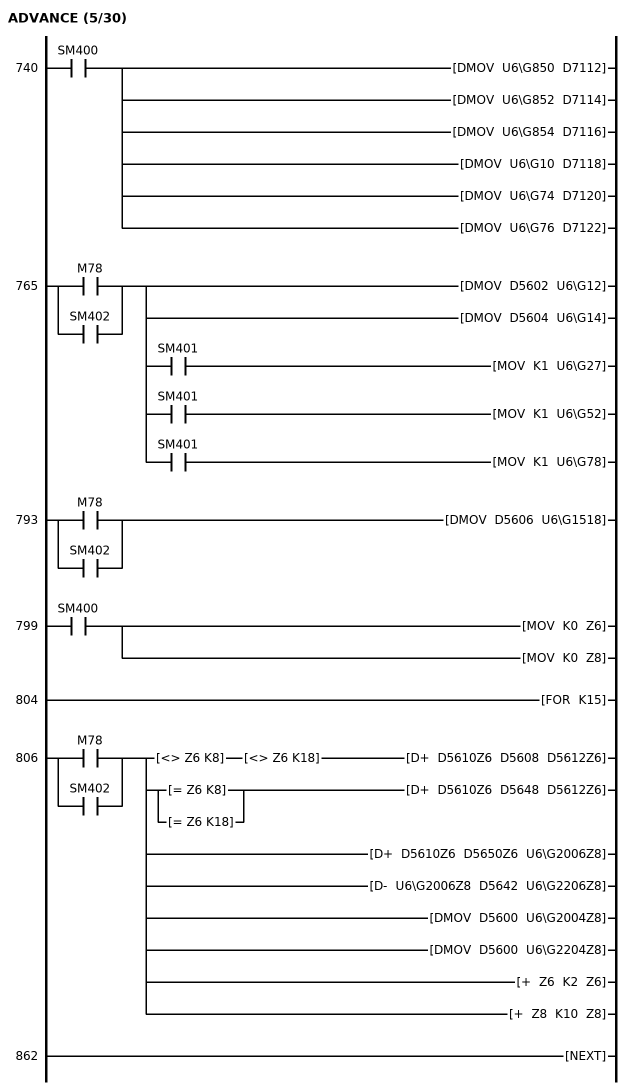
[picture p360: ladder of ADVANCE, rungs at steps 740 to 862]
740   LD      SM400
      DMOV    U6\G850 D7112
      DMOV    U6\G852 D7114
      DMOV    U6\G854 D7116
      DMOV    U6\G10 D7118
      DMOV    U6\G74 D7120
      DMOV    U6\G76 D7122
765   LD      M78
      OR      SM402
      DMOV    D5602 U6\G12
      DMOV    D5604 U6\G14
      MPS
      AND     SM401
      MOV     K1 U6\G27
      MRD
      AND     SM401
      MOV     K1 U6\G52
      MPP
      AND     SM401
      MOV     K1 U6\G78
793   LD      M78
      OR      SM402
      DMOV    D5606 U6\G1518
799   LD      SM400
      MOV     K0 Z6
      MOV     K0 Z8
804   FOR     K15
806   LD      M78
      OR      SM402
      MPS
      AND<>   Z6 K8
      AND<>   Z6 K18
      D+      D5610Z6 D5608 D5612Z6
      MRD
      LD=     Z6 K8
      OR=     Z6 K18
      ANB
      D+      D5610Z6 D5648 D5612Z6
      MPP
      D+      D5610Z6 D5650Z6 U6\G2006Z8
      D-      U6\G2006Z8 D5642 U6\G2206Z8
      DMOV    D5600 U6\G2004Z8
      DMOV    D5600 U6\G2204Z8
      +       Z6 K2 Z6
      +       Z8 K10 Z8
862   NEXT
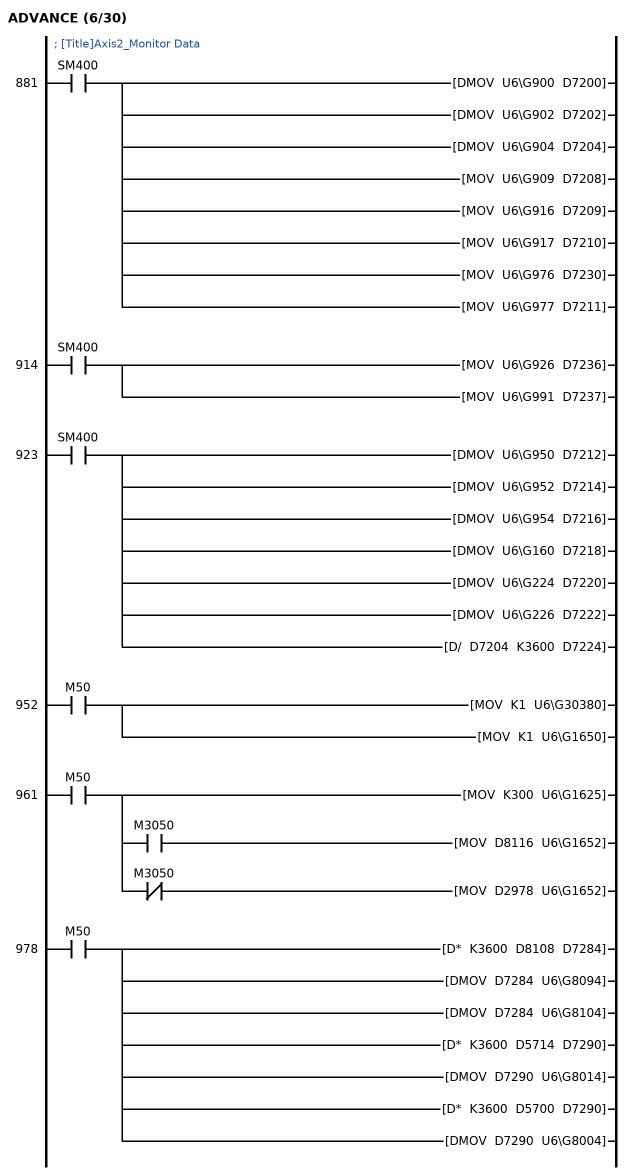
; 
; [Title]Axis2_Monitor Data
; 
; 
881   LD      SM400
      DMOV    U6\G900 D7200
      DMOV    U6\G902 D7202
      DMOV    U6\G904 D7204
      MOV     U6\G909 D7208
      MOV     U6\G916 D7209
      MOV     U6\G917 D7210
      MOV     U6\G976 D7230
      MOV     U6\G977 D7211
914   LD      SM400
      MOV     U6\G926 D7236
      MOV     U6\G991 D7237
923   LD      SM400
      DMOV    U6\G950 D7212
      DMOV    U6\G952 D7214
      DMOV    U6\G954 D7216
      DMOV    U6\G160 D7218
      DMOV    U6\G224 D7220
      DMOV    U6\G226 D7222
      D/      D7204 K3600 D7224
952   LD      M50
      MOV     K1 U6\G30380
      MOV     K1 U6\G1650
961   LD      M50
      MOV     K300 U6\G1625
      MPS
      AND     M3050
      MOV     D8116 U6\G1652
      MPP
      ANI     M3050
      MOV     D2978 U6\G1652
978   LD      M50
      D*      K3600 D8108 D7284
      DMOV    D7284 U6\G8094
      DMOV    D7284 U6\G8104
      D*      K3600 D5714 D7290
      DMOV    D7290 U6\G8014
      D*      K3600 D5700 D7290
      DMOV    D7290 U6\G8004
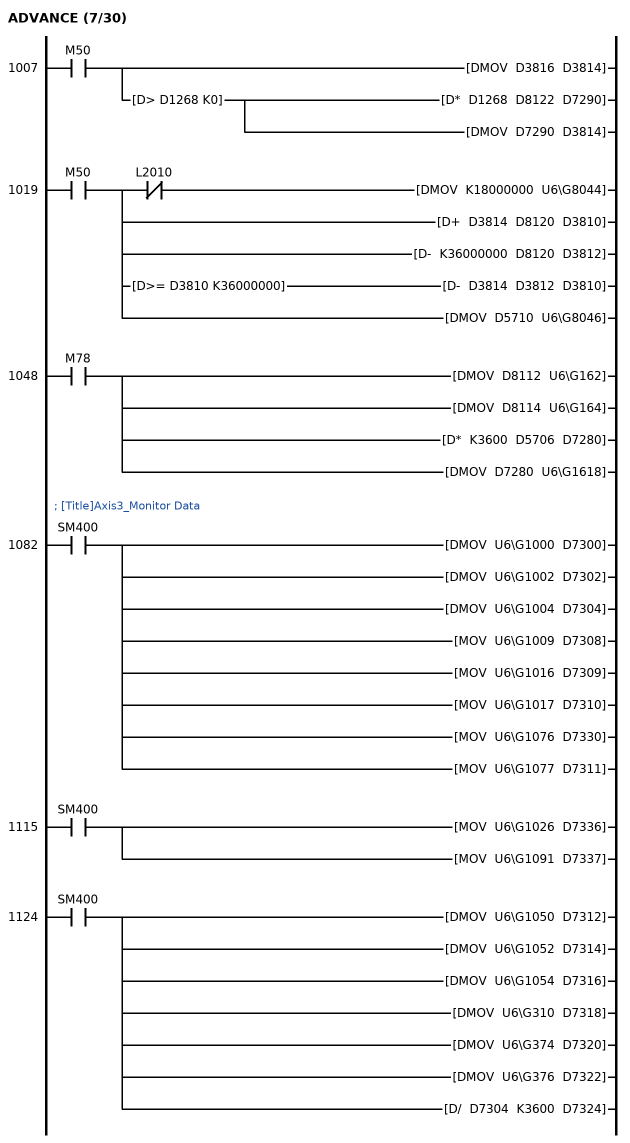
1007  LD      M50
      DMOV    D3816 D3814
      ANDD>   D1268 K0
      D*      D1268 D8122 D7290
      DMOV    D7290 D3814
1019  LD      M50
      MPS
      ANI     L2010
      DMOV    K18000000 U6\G8044
      MPP
      D+      D3814 D8120 D3810
      D-      K36000000 D8120 D3812
      MPS
      ANDD>=  D3810 K36000000
      D-      D3814 D3812 D3810
      MPP
      DMOV    D5710 U6\G8046
1048  LD      M78
      DMOV    D8112 U6\G162
      DMOV    D8114 U6\G164
      D*      K3600 D5706 D7280
      DMOV    D7280 U6\G1618
; 
; [Title]Axis3_Monitor Data
; 
1082  LD      SM400
      DMOV    U6\G1000 D7300
      DMOV    U6\G1002 D7302
      DMOV    U6\G1004 D7304
      MOV     U6\G1009 D7308
      MOV     U6\G1016 D7309
      MOV     U6\G1017 D7310
      MOV     U6\G1076 D7330
      MOV     U6\G1077 D7311
1115  LD      SM400
      MOV     U6\G1026 D7336
      MOV     U6\G1091 D7337
1124  LD      SM400
      DMOV    U6\G1050 D7312
      DMOV    U6\G1052 D7314
      DMOV    U6\G1054 D7316
      DMOV    U6\G310 D7318
      DMOV    U6\G374 D7320
      DMOV    U6\G376 D7322
      D/      D7304 K3600 D7324
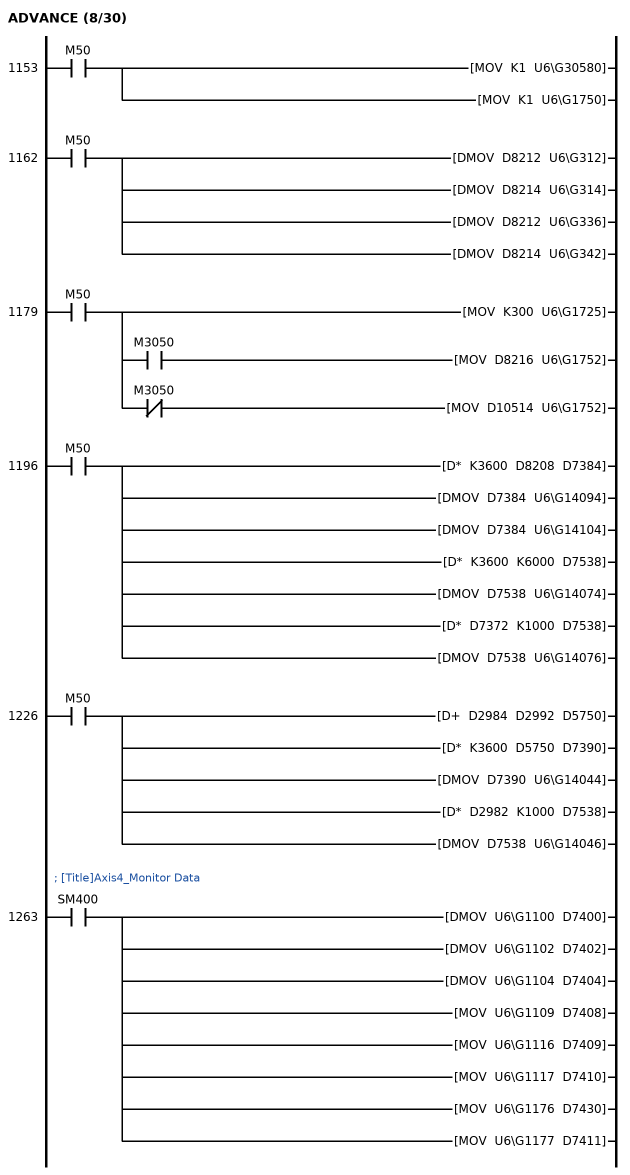
1153  LD      M50
      MOV     K1 U6\G30580
      MOV     K1 U6\G1750
1162  LD      M50
      DMOV    D8212 U6\G312
      DMOV    D8214 U6\G314
      DMOV    D8212 U6\G336
      DMOV    D8214 U6\G342
1179  LD      M50
      MOV     K300 U6\G1725
      MPS
      AND     M3050
      MOV     D8216 U6\G1752
      MPP
      ANI     M3050
      MOV     D10514 U6\G1752
1196  LD      M50
      D*      K3600 D8208 D7384
      DMOV    D7384 U6\G14094
      DMOV    D7384 U6\G14104
      D*      K3600 K6000 D7538
      DMOV    D7538 U6\G14074
      D*      D7372 K1000 D7538
      DMOV    D7538 U6\G14076
1226  LD      M50
      D+      D2984 D2992 D5750
      D*      K3600 D5750 D7390
      DMOV    D7390 U6\G14044
      D*      D2982 K1000 D7538
      DMOV    D7538 U6\G14046
; [Title]Axis4_Monitor Data
; 
; 
1263  LD      SM400
      DMOV    U6\G1100 D7400
      DMOV    U6\G1102 D7402
      DMOV    U6\G1104 D7404
      MOV     U6\G1109 D7408
      MOV     U6\G1116 D7409
      MOV     U6\G1117 D7410
      MOV     U6\G1176 D7430
      MOV     U6\G1177 D7411
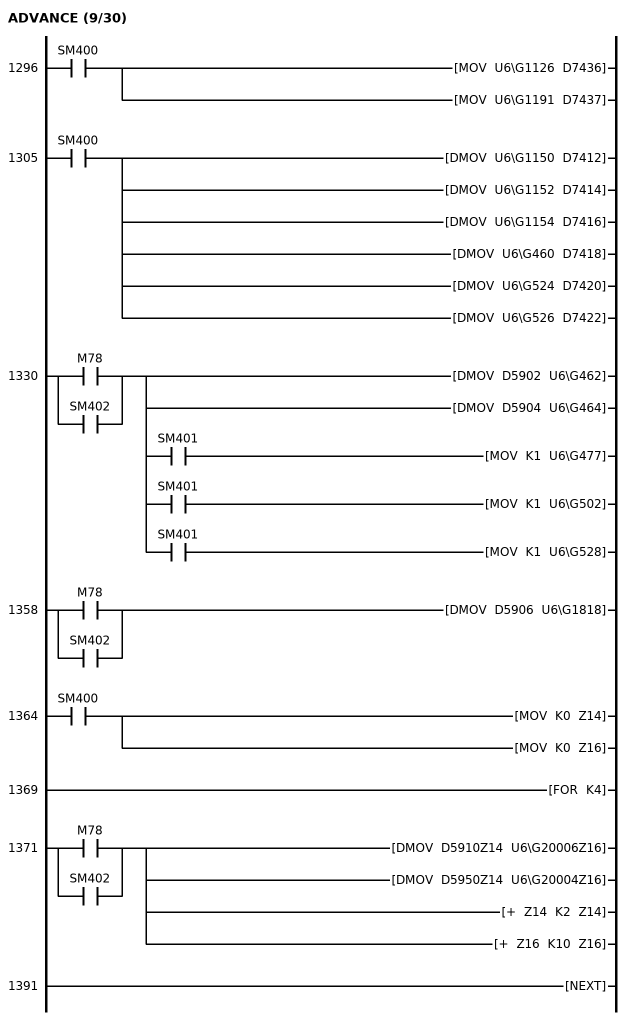
1296  LD      SM400
      MOV     U6\G1126 D7436
      MOV     U6\G1191 D7437
1305  LD      SM400
      DMOV    U6\G1150 D7412
      DMOV    U6\G1152 D7414
      DMOV    U6\G1154 D7416
      DMOV    U6\G460 D7418
      DMOV    U6\G524 D7420
      DMOV    U6\G526 D7422
1330  LD      M78
      OR      SM402
      DMOV    D5902 U6\G462
      DMOV    D5904 U6\G464
      MPS
      AND     SM401
      MOV     K1 U6\G477
      MRD
      AND     SM401
      MOV     K1 U6\G502
      MPP
      AND     SM401
      MOV     K1 U6\G528
1358  LD      M78
      OR      SM402
      DMOV    D5906 U6\G1818
1364  LD      SM400
      MOV     K0 Z14
      MOV     K0 Z16
1369  FOR     K4
1371  LD      M78
      OR      SM402
      DMOV    D5910Z14 U6\G20006Z16
      DMOV    D5950Z14 U6\G20004Z16
      +       Z14 K2 Z14
      +       Z16 K10 Z16
1391  NEXT
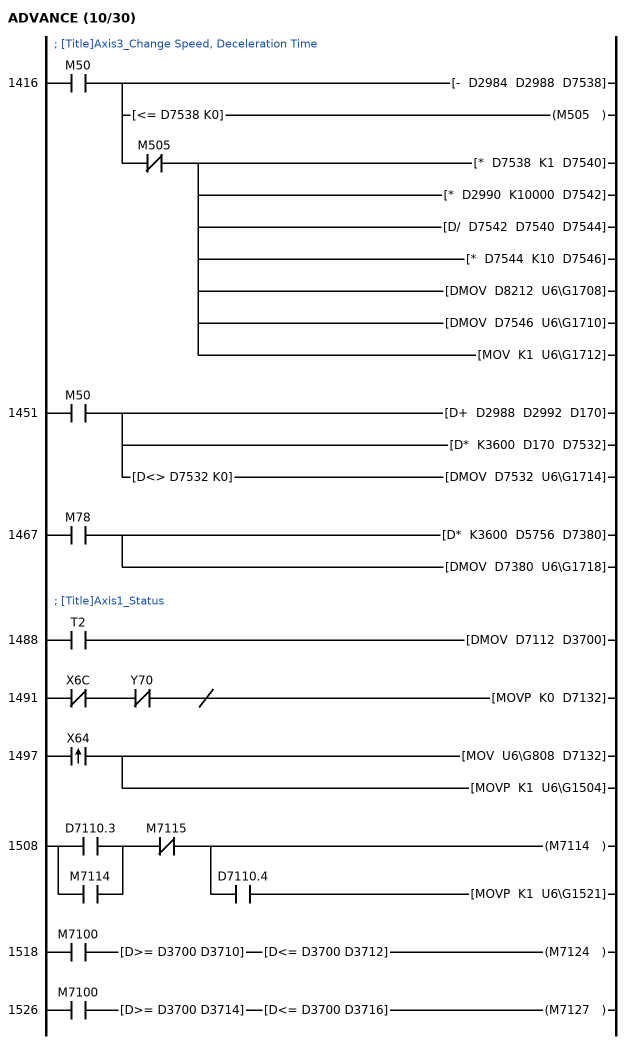
; [Title]Axis3_Change Speed, Deceleration Time
1416  LD      M50
      -       D2984 D2988 D7538
      MPS
      AND<=   D7538 K0
      OUT     M505
      MPP
      ANI     M505
      *       D7538 K1 D7540
      *       D2990 K10000 D7542
      D/      D7542 D7540 D7544
      *       D7544 K10 D7546
      DMOV    D8212 U6\G1708
      DMOV    D7546 U6\G1710
      MOV     K1 U6\G1712
1451  LD      M50
      D+      D2988 D2992 D170
      D*      K3600 D170 D7532
      ANDD<>  D7532 K0
      DMOV    D7532 U6\G1714
1467  LD      M78
      D*      K3600 D5756 D7380
      DMOV    D7380 U6\G1718
; [Title]Axis1_Status
1488  LD      T2
      DMOV    D7112 D3700
1491  LDI     X6C
      ANI     Y70
      INV
      MOVP    K0 D7132
1497  LDP     X64
      MOV     U6\G808 D7132
      MOVP    K1 U6\G1504
1508  LD      D7110.3
      OR      M7114
      ANI     M7115
      OUT     M7114
      AND     D7110.4
      MOVP    K1 U6\G1521
1518  LD      M7100
      ANDD>=  D3700 D3710
      ANDD<=  D3700 D3712
      OUT     M7124
1526  LD      M7100
      ANDD>=  D3700 D3714
      ANDD<=  D3700 D3716
      OUT     M7127
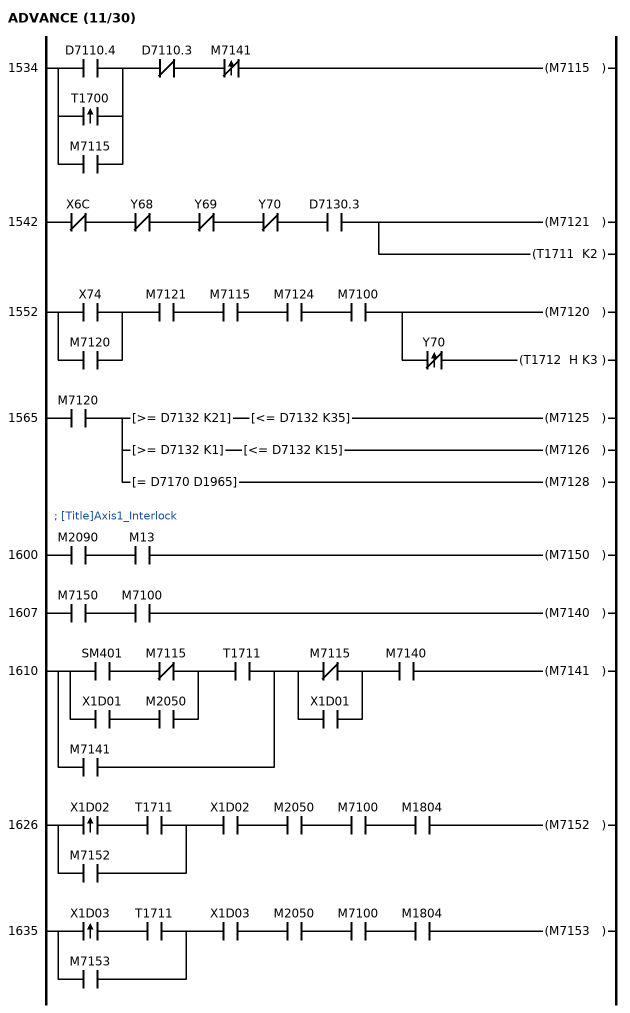
1534  LD      D7110.4
      ORP     T1700
      OR      M7115
      ANI     D7110.3
      ANDPI   M7141
      OUT     M7115
1542  LDI     X6C
      ANI     Y68
      ANI     Y69
      ANI     Y70
      AND     D7130.3
      OUT     M7121
      OUT     T1711 K2
1552  LD      X74
      OR      M7120
      AND     M7121
      AND     M7115
      AND     M7124
      AND     M7100
      OUT     M7120
      ANDPI   Y70
      OUTH    T1712 K3
1565  LD      M7120
      MPS
      AND>=   D7132 K21
      AND<=   D7132 K35
      OUT     M7125
      MRD
      AND>=   D7132 K1
      AND<=   D7132 K15
      OUT     M7126
      MPP
      AND=    D7170 D1965
      OUT     M7128
; [Title]Axis1_Interlock
1600  LD      M2090
      AND     M13
      OUT     M7150
; 
; 
; 
; 
1607  LD      M7150
      AND     M7100
      OUT     M7140
1610  LD      SM401
      ANI     M7115
      LD      X1D01
      AND     M2050
      ORB
      AND     T1711
      OR      M7141
      LDI     M7115
      OR      X1D01
      ANB
      AND     M7140
      OUT     M7141
; 
; 
; 
; 
1626  LDP     X1D02
      AND     T1711
      OR      M7152
      AND     X1D02
      AND     M2050
      AND     M7100
      AND     M1804
      OUT     M7152
1635  LDP     X1D03
      AND     T1711
      OR      M7153
      AND     X1D03
      AND     M2050
      AND     M7100
      AND     M1804
      OUT     M7153
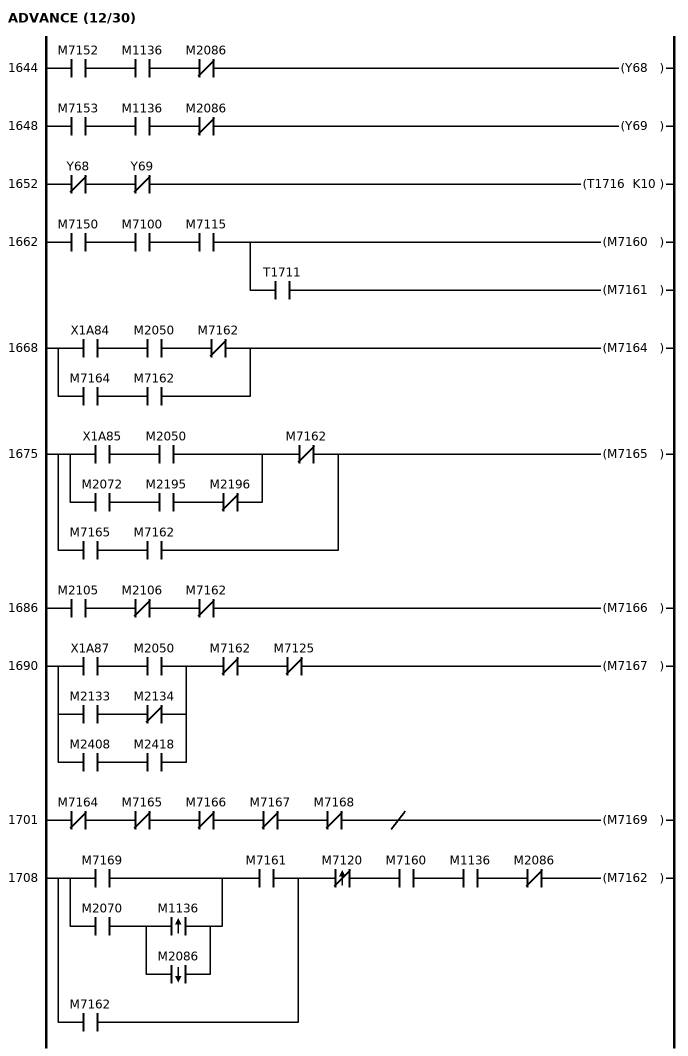
1644  LD      M7152
      AND     M1136
      ANI     M2086
      OUT     Y68
1648  LD      M7153
      AND     M1136
      ANI     M2086
      OUT     Y69
1652  LDI     Y68
      ANI     Y69
      OUT     T1716 K10
; 
; 
; 
; 
1662  LD      M7150
      AND     M7100
      AND     M7115
      OUT     M7160
      AND     T1711
      OUT     M7161
1668  LD      X1A84
      AND     M2050
      ANI     M7162
      LD      M7164
      AND     M7162
      ORB
      OUT     M7164
1675  LD      X1A85
      AND     M2050
      LD      M2072
      AND     M2195
      ANI     M2196
      ORB
      ANI     M7162
      LD      M7165
      AND     M7162
      ORB
      OUT     M7165
1686  LD      M2105
      ANI     M2106
      ANI     M7162
      OUT     M7166
1690  LD      X1A87
      AND     M2050
      LD      M2133
      ANI     M2134
      ORB
      LD      M2408
      AND     M2418
      ORB
      ANI     M7162
      ANI     M7125
      OUT     M7167
1701  LDI     M7164
      ANI     M7165
      ANI     M7166
      ANI     M7167
      ANI     M7168
      INV
      OUT     M7169
1708  LD      M7169
      LD      M2070
      LDP     M1136
      ORF     M2086
      ANB
      ORB
      AND     M7161
      OR      M7162
      ANDPI   M7120
      AND     M7160
      AND     M1136
      ANI     M2086
      OUT     M7162
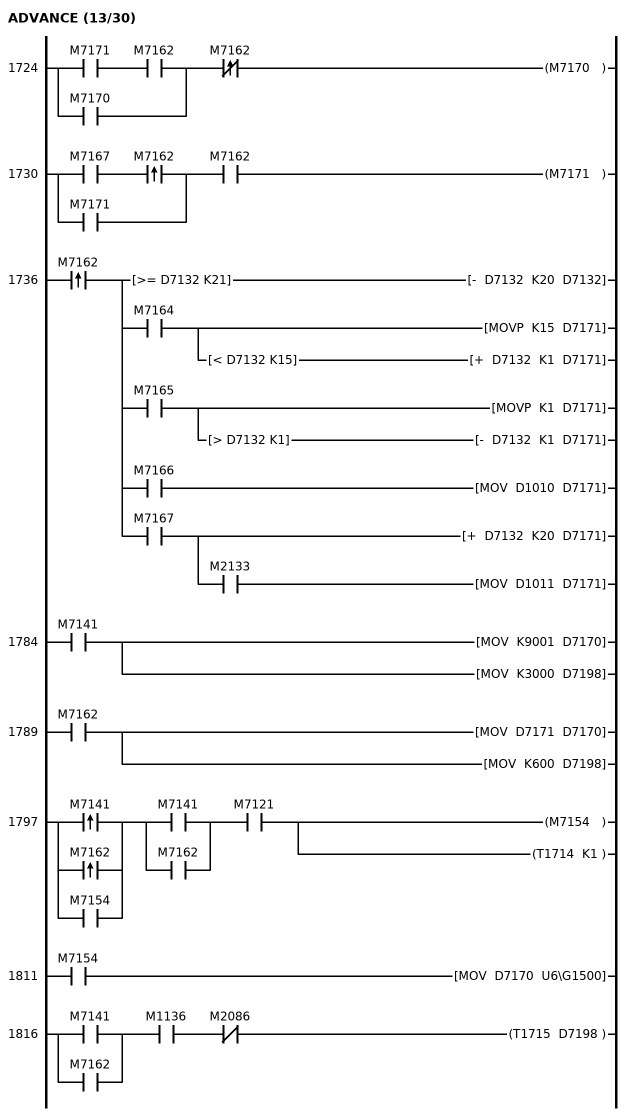
1724  LD      M7171
      AND     M7162
      OR      M7170
      ANDPI   M7162
      OUT     M7170
1730  LD      M7167
      ANDP    M7162
      OR      M7171
      AND     M7162
      OUT     M7171
1736  LDP     M7162
      MPS
      AND>=   D7132 K21
      -       D7132 K20 D7132
      MRD
      AND     M7164
      MOVP    K15 D7171
      AND<    D7132 K15
      +       D7132 K1 D7171
      MRD
      AND     M7165
      MOVP    K1 D7171
      AND>    D7132 K1
      -       D7132 K1 D7171
      MRD
      AND     M7166
      MOV     D1010 D7171
      MPP
      AND     M7167
      +       D7132 K20 D7171
      AND     M2133
      MOV     D1011 D7171
; 
; 
; 
; 
1784  LD      M7141
      MOV     K9001 D7170
      MOV     K3000 D7198
1789  LD      M7162
      MOV     D7171 D7170
      MOV     K600 D7198
; 
; 
; 
1797  LDP     M7141
      ORP     M7162
      OR      M7154
      LD      M7141
      OR      M7162
      ANB
      AND     M7121
      OUT     M7154
      OUT     T1714 K1
1811  LD      M7154
      MOV     D7170 U6\G1500
1816  LD      M7141
      OR      M7162
      AND     M1136
      ANI     M2086
      OUT     T1715 D7198
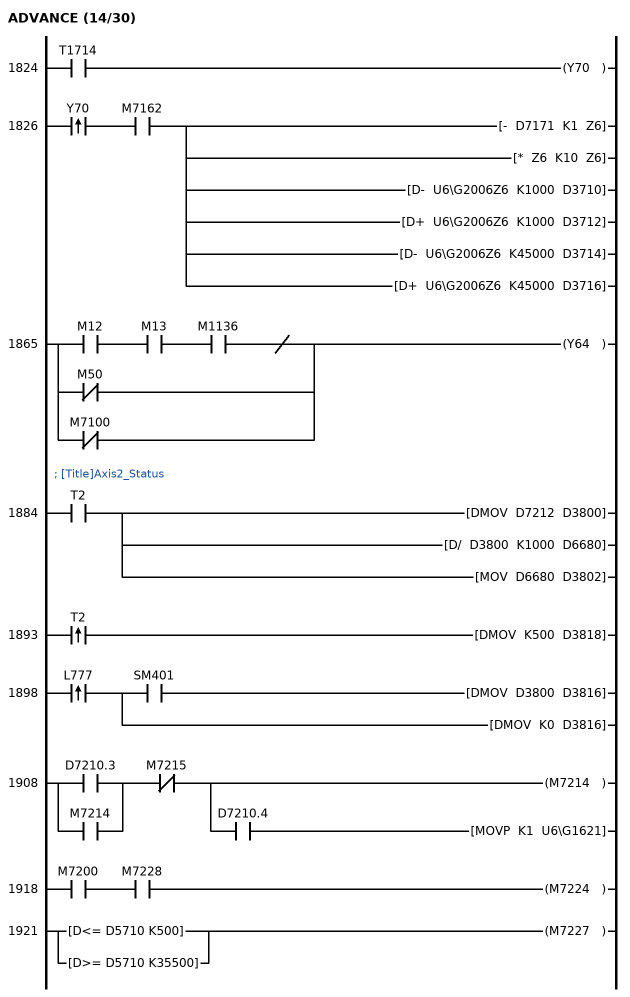
1824  LD      T1714
      OUT     Y70
1826  LDP     Y70
      AND     M7162
      -       D7171 K1 Z6
      *       Z6 K10 Z6
      D-      U6\G2006Z6 K1000 D3710
      D+      U6\G2006Z6 K1000 D3712
      D-      U6\G2006Z6 K45000 D3714
      D+      U6\G2006Z6 K45000 D3716
; 
; 
; 
1865  LD      M12
      AND     M13
      AND     M1136
      INV
      ORI     M50
      ORI     M7100
      OUT     Y64
; [Title]Axis2_Status
1884  LD      T2
      DMOV    D7212 D3800
      D/      D3800 K1000 D6680
      MOV     D6680 D3802
1893  LDP     T2
      DMOV    K500 D3818
1898  LDP     L777
      MPS
      AND     SM401
      DMOV    D3800 D3816
      MPP
      DMOV    K0 D3816
1908  LD      D7210.3
      OR      M7214
      ANI     M7215
      OUT     M7214
      AND     D7210.4
      MOVP    K1 U6\G1621
1918  LD      M7200
      AND     M7228
      OUT     M7224
1921  LDD<=   D5710 K500
      ORD>=   D5710 K35500
      OUT     M7227
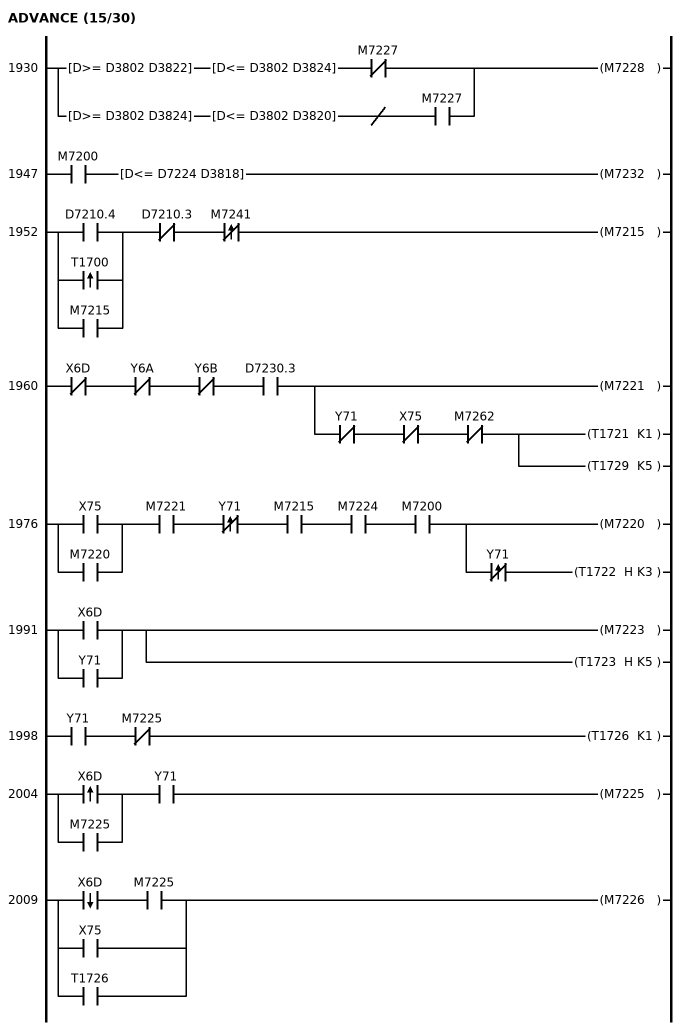
1930  LDD>=   D3802 D3822
      ANDD<=  D3802 D3824
      ANI     M7227
      LDD>=   D3802 D3824
      ANDD<=  D3802 D3820
      INV
      AND     M7227
      ORB
      OUT     M7228
1947  LD      M7200
      ANDD<=  D7224 D3818
      OUT     M7232
1952  LD      D7210.4
      ORP     T1700
      OR      M7215
      ANI     D7210.3
      ANDPI   M7241
      OUT     M7215
1960  LDI     X6D
      ANI     Y6A
      ANI     Y6B
      AND     D7230.3
      OUT     M7221
      ANI     Y71
      ANI     X75
      ANI     M7262
      OUT     T1721 K1
      OUT     T1729 K5
1976  LD      X75
      OR      M7220
      AND     M7221
      ANDPI   Y71
      AND     M7215
      AND     M7224
      AND     M7200
      OUT     M7220
      ANDPI   Y71
      OUTH    T1722 K3
1991  LD      X6D
      OR      Y71
      OUT     M7223
      OUTH    T1723 K5
1998  LD      Y71
      ANI     M7225
      OUT     T1726 K1
2004  LDP     X6D
      OR      M7225
      AND     Y71
      OUT     M7225
2009  LDF     X6D
      AND     M7225
      OR      X75
      OR      T1726
      OUT     M7226
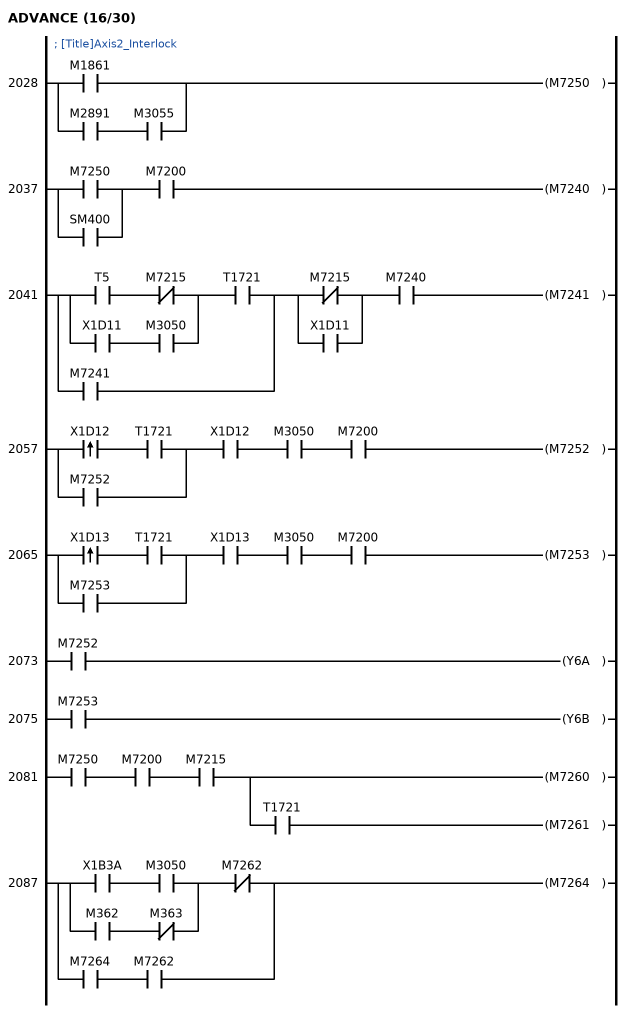
; [Title]Axis2_Interlock
2028  LD      M1861
      LD      M2891
      AND     M3055
      ORB
      OUT     M7250
; 
; 
; 
; 
2037  LD      M7250
      OR      SM400
      AND     M7200
      OUT     M7240
2041  LD      T5
      ANI     M7215
      LD      X1D11
      AND     M3050
      ORB
      AND     T1721
      OR      M7241
      LDI     M7215
      OR      X1D11
      ANB
      AND     M7240
      OUT     M7241
; 
; 
; 
; 
2057  LDP     X1D12
      AND     T1721
      OR      M7252
      AND     X1D12
      AND     M3050
      AND     M7200
      OUT     M7252
2065  LDP     X1D13
      AND     T1721
      OR      M7253
      AND     X1D13
      AND     M3050
      AND     M7200
      OUT     M7253
2073  LD      M7252
      OUT     Y6A
2075  LD      M7253
      OUT     Y6B
; 
; 
; 
; 
2081  LD      M7250
      AND     M7200
      AND     M7215
      OUT     M7260
      AND     T1721
      OUT     M7261
2087  LD      X1B3A
      AND     M3050
      LD      M362
      ANI     M363
      ORB
      ANI     M7262
      LD      M7264
      AND     M7262
      ORB
      OUT     M7264
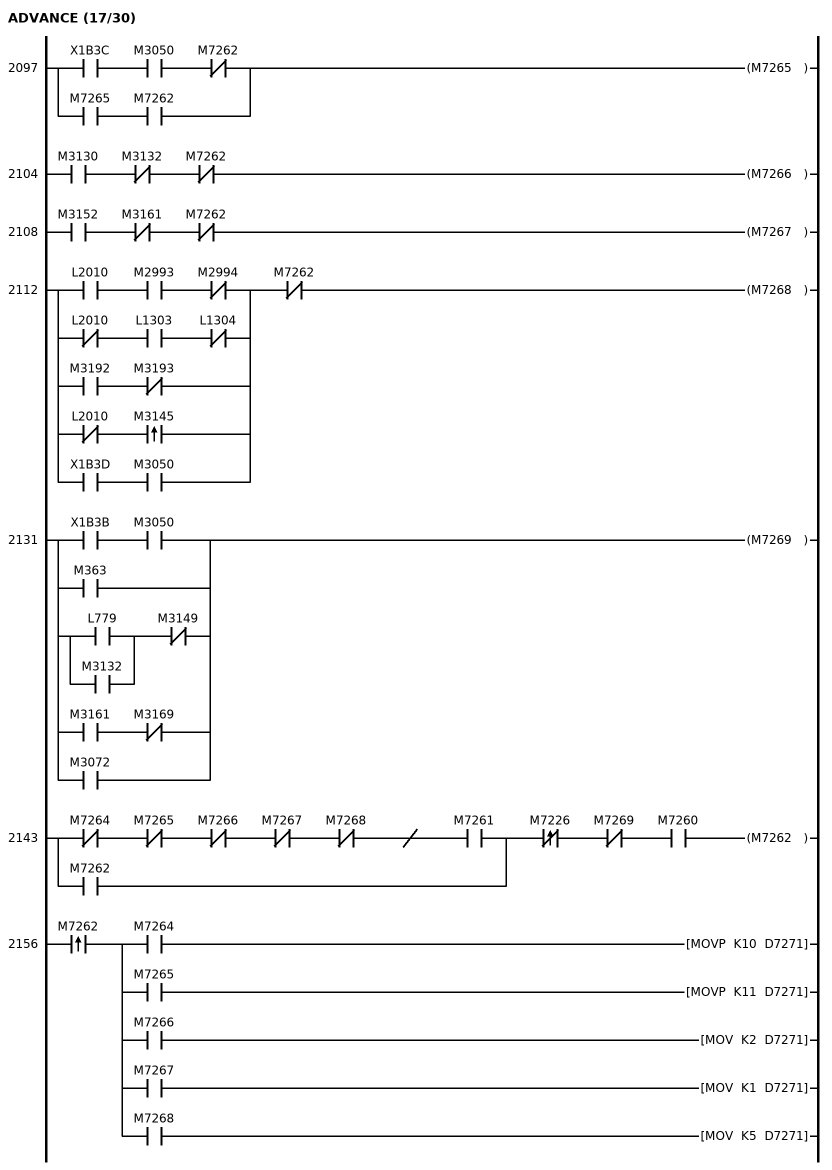
2097  LD      X1B3C
      AND     M3050
      ANI     M7262
      LD      M7265
      AND     M7262
      ORB
      OUT     M7265
2104  LD      M3130
      ANI     M3132
      ANI     M7262
      OUT     M7266
2108  LD      M3152
      ANI     M3161
      ANI     M7262
      OUT     M7267
2112  LD      L2010
      AND     M2993
      ANI     M2994
      LDI     L2010
      AND     L1303
      ANI     L1304
      ORB
      LD      M3192
      ANI     M3193
      ORB
      LDI     L2010
      ANDP    M3145
      ORB
      LD      X1B3D
      AND     M3050
      ORB
      ANI     M7262
      OUT     M7268
2131  LD      X1B3B
      AND     M3050
      OR      M363
      LD      L779
      OR      M3132
      ANI     M3149
      ORB
      LD      M3161
      ANI     M3169
      ORB
      OR      M3072
      OUT     M7269
2143  LDI     M7264
      ANI     M7265
      ANI     M7266
      ANI     M7267
      ANI     M7268
      INV
      AND     M7261
      OR      M7262
      ANDPI   M7226
      ANI     M7269
      AND     M7260
      OUT     M7262
2156  LDP     M7262
      MPS
      AND     M7264
      MOVP    K10 D7271
      MRD
      AND     M7265
      MOVP    K11 D7271
      MRD
      AND     M7266
      MOV     K2 D7271
      MRD
      AND     M7267
      MOV     K1 D7271
      MPP
      AND     M7268
      MOV     K5 D7271
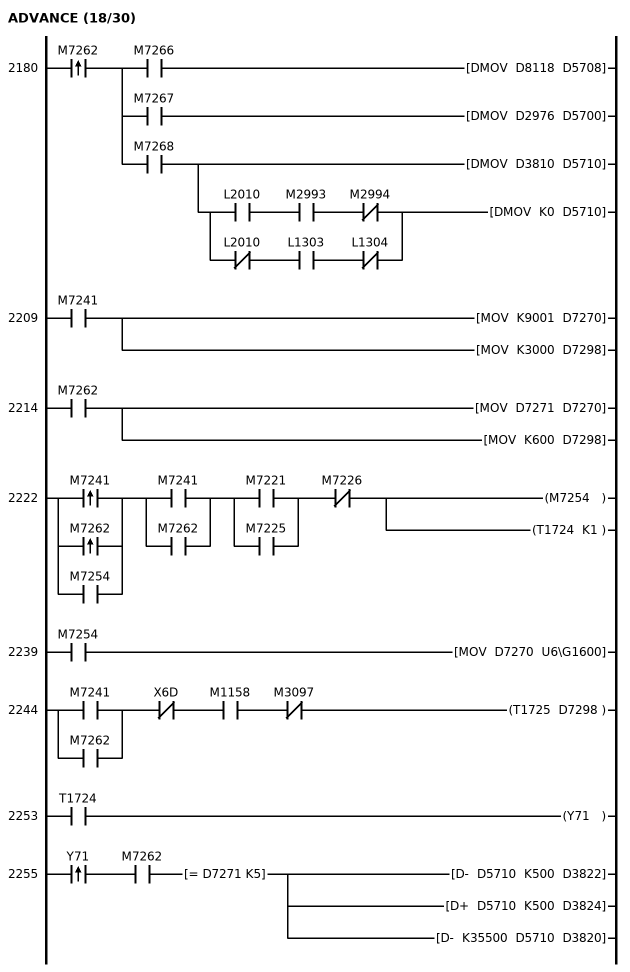
2180  LDP     M7262
      MPS
      AND     M7266
      DMOV    D8118 D5708
      MRD
      AND     M7267
      DMOV    D2976 D5700
      MPP
      AND     M7268
      DMOV    D3810 D5710
      LD      L2010
      AND     M2993
      ANI     M2994
      LDI     L2010
      AND     L1303
      ANI     L1304
      ORB
      ANB
      DMOV    K0 D5710
; 
; 
; 
; 
2209  LD      M7241
      MOV     K9001 D7270
      MOV     K3000 D7298
2214  LD      M7262
      MOV     D7271 D7270
      MOV     K600 D7298
; 
; 
; 
2222  LDP     M7241
      ORP     M7262
      OR      M7254
      LD      M7241
      OR      M7262
      ANB
      LD      M7221
      OR      M7225
      ANB
      ANI     M7226
      OUT     M7254
      OUT     T1724 K1
2239  LD      M7254
      MOV     D7270 U6\G1600
2244  LD      M7241
      OR      M7262
      ANI     X6D
      AND     M1158
      ANI     M3097
      OUT     T1725 D7298
2253  LD      T1724
      OUT     Y71
2255  LDP     Y71
      AND     M7262
      AND=    D7271 K5
      D-      D5710 K500 D3822
      D+      D5710 K500 D3824
      D-      K35500 D5710 D3820
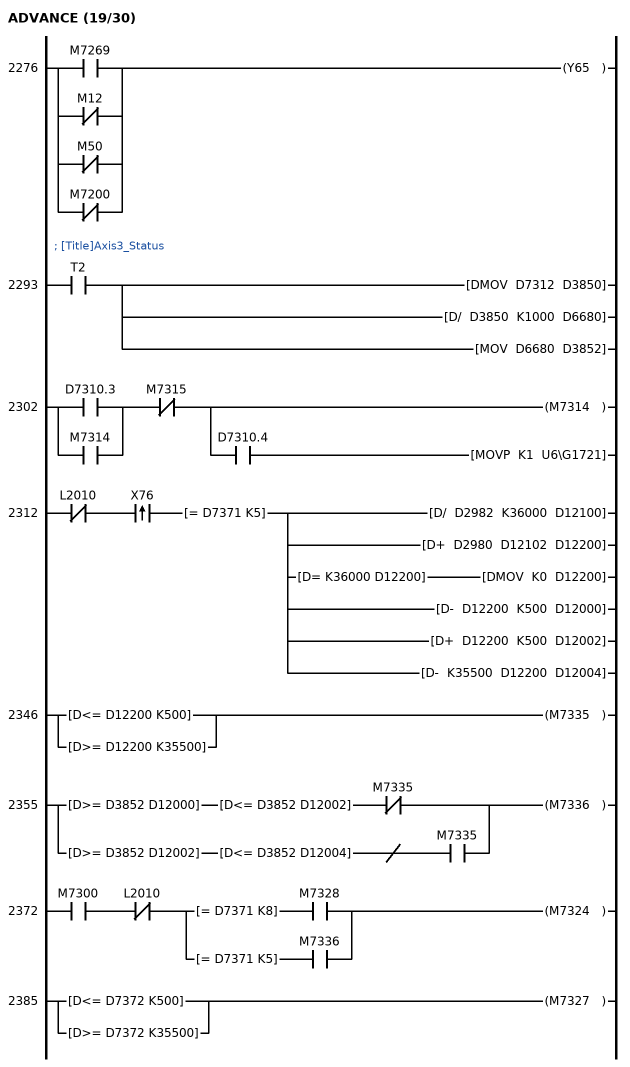
; 
; 
; 
2276  LD      M7269
      ORI     M12
      ORI     M50
      ORI     M7200
      OUT     Y65
; [Title]Axis3_Status
2293  LD      T2
      DMOV    D7312 D3850
      D/      D3850 K1000 D6680
      MOV     D6680 D3852
2302  LD      D7310.3
      OR      M7314
      ANI     M7315
      OUT     M7314
      AND     D7310.4
      MOVP    K1 U6\G1721
2312  LDI     L2010
      ANDP    X76
      AND=    D7371 K5
      D/      D2982 K36000 D12100
      D+      D2980 D12102 D12200
      MPS
      ANDD=   K36000 D12200
      DMOV    K0 D12200
      MPP
      D-      D12200 K500 D12000
      D+      D12200 K500 D12002
      D-      K35500 D12200 D12004
2346  LDD<=   D12200 K500
      ORD>=   D12200 K35500
      OUT     M7335
2355  LDD>=   D3852 D12000
      ANDD<=  D3852 D12002
      ANI     M7335
      LDD>=   D3852 D12002
      ANDD<=  D3852 D12004
      INV
      AND     M7335
      ORB
      OUT     M7336
2372  LD      M7300
      ANI     L2010
      LD=     D7371 K8
      AND     M7328
      LD=     D7371 K5
      AND     M7336
      ORB
      ANB
      OUT     M7324
2385  LDD<=   D7372 K500
      ORD>=   D7372 K35500
      OUT     M7327
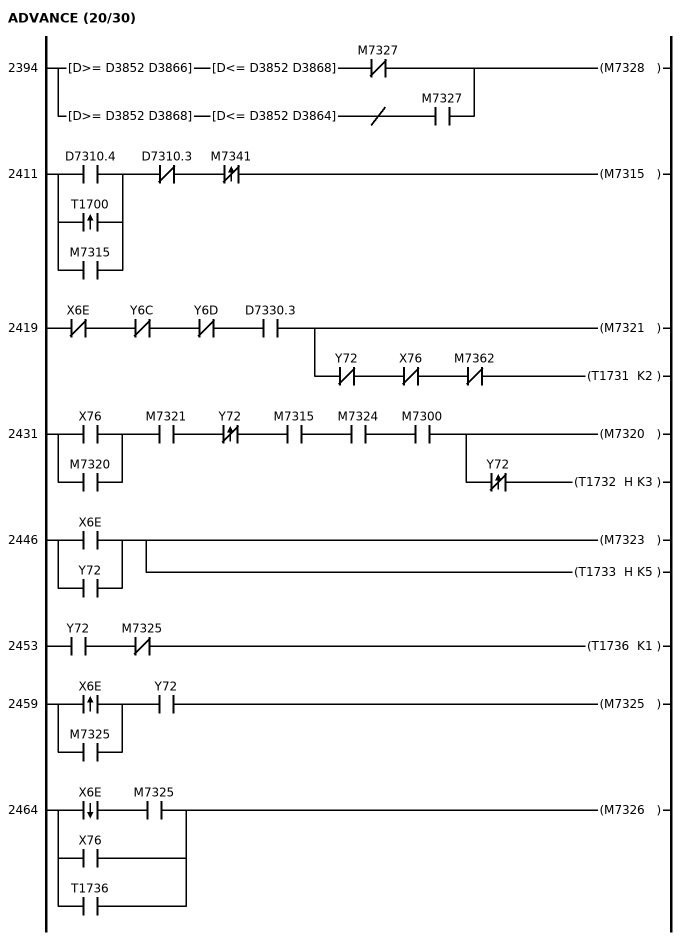
2394  LDD>=   D3852 D3866
      ANDD<=  D3852 D3868
      ANI     M7327
      LDD>=   D3852 D3868
      ANDD<=  D3852 D3864
      INV
      AND     M7327
      ORB
      OUT     M7328
2411  LD      D7310.4
      ORP     T1700
      OR      M7315
      ANI     D7310.3
      ANDPI   M7341
      OUT     M7315
2419  LDI     X6E
      ANI     Y6C
      ANI     Y6D
      AND     D7330.3
      OUT     M7321
      ANI     Y72
      ANI     X76
      ANI     M7362
      OUT     T1731 K2
2431  LD      X76
      OR      M7320
      AND     M7321
      ANDPI   Y72
      AND     M7315
      AND     M7324
      AND     M7300
      OUT     M7320
      ANDPI   Y72
      OUTH    T1732 K3
2446  LD      X6E
      OR      Y72
      OUT     M7323
      OUTH    T1733 K5
2453  LD      Y72
      ANI     M7325
      OUT     T1736 K1
2459  LDP     X6E
      OR      M7325
      AND     Y72
      OUT     M7325
2464  LDF     X6E
      AND     M7325
      OR      X76
      OR      T1736
      OUT     M7326
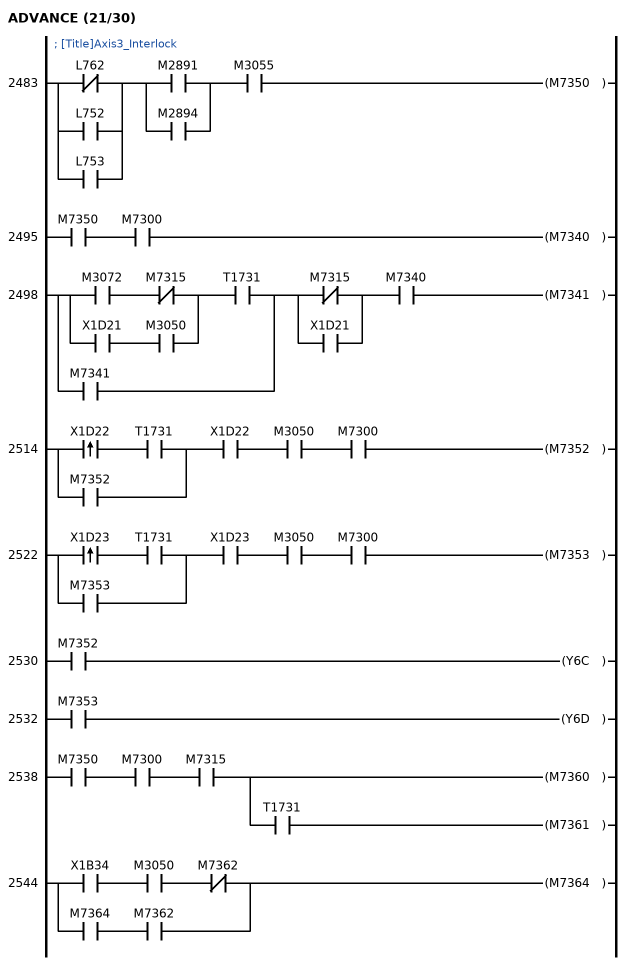
; [Title]Axis3_Interlock
2483  LDI     L762
      OR      L752
      OR      L753
      LD      M2891
      OR      M2894
      ANB
      AND     M3055
      OUT     M7350
; 
; 
; 
; 
2495  LD      M7350
      AND     M7300
      OUT     M7340
2498  LD      M3072
      ANI     M7315
      LD      X1D21
      AND     M3050
      ORB
      AND     T1731
      OR      M7341
      LDI     M7315
      OR      X1D21
      ANB
      AND     M7340
      OUT     M7341
; 
; 
; 
; 
2514  LDP     X1D22
      AND     T1731
      OR      M7352
      AND     X1D22
      AND     M3050
      AND     M7300
      OUT     M7352
2522  LDP     X1D23
      AND     T1731
      OR      M7353
      AND     X1D23
      AND     M3050
      AND     M7300
      OUT     M7353
2530  LD      M7352
      OUT     Y6C
2532  LD      M7353
      OUT     Y6D
; 
; 
; 
; 
2538  LD      M7350
      AND     M7300
      AND     M7315
      OUT     M7360
      AND     T1731
      OUT     M7361
2544  LD      X1B34
      AND     M3050
      ANI     M7362
      LD      M7364
      AND     M7362
      ORB
      OUT     M7364
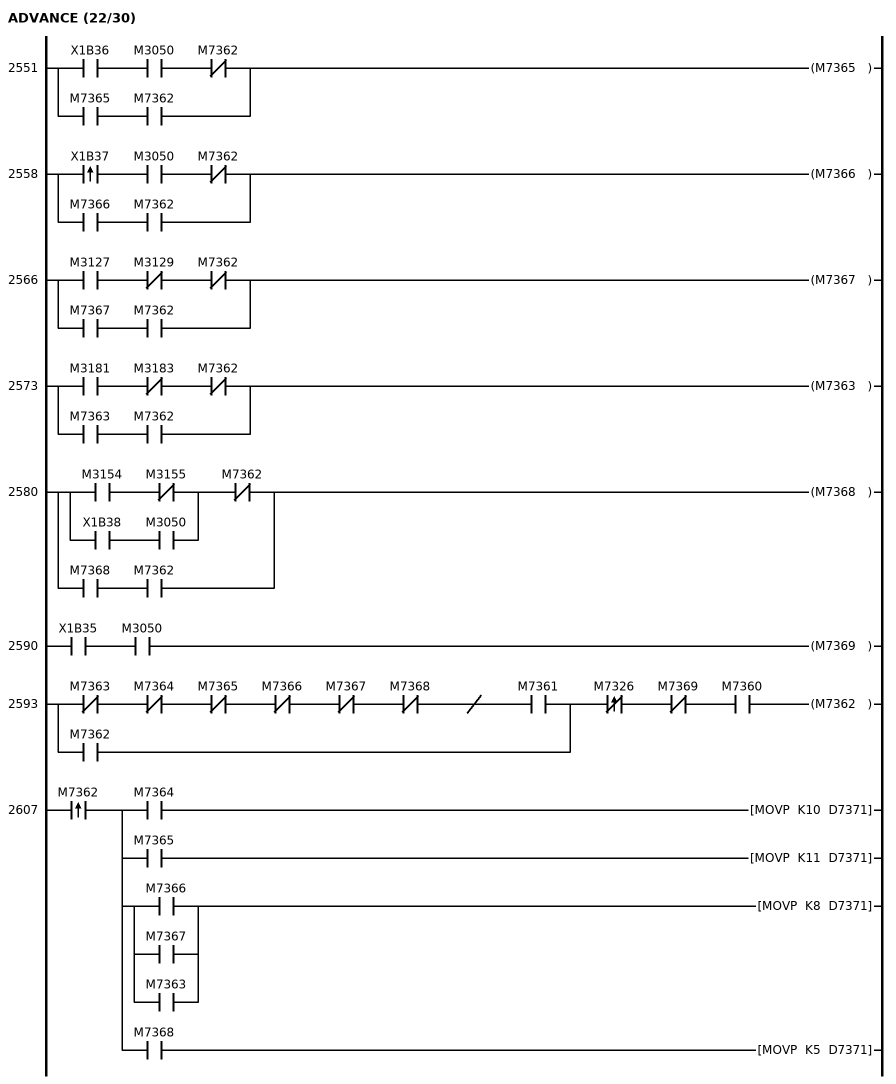
2551  LD      X1B36
      AND     M3050
      ANI     M7362
      LD      M7365
      AND     M7362
      ORB
      OUT     M7365
2558  LDP     X1B37
      AND     M3050
      ANI     M7362
      LD      M7366
      AND     M7362
      ORB
      OUT     M7366
2566  LD      M3127
      ANI     M3129
      ANI     M7362
      LD      M7367
      AND     M7362
      ORB
      OUT     M7367
2573  LD      M3181
      ANI     M3183
      ANI     M7362
      LD      M7363
      AND     M7362
      ORB
      OUT     M7363
2580  LD      M3154
      ANI     M3155
      LD      X1B38
      AND     M3050
      ORB
      ANI     M7362
      LD      M7368
      AND     M7362
      ORB
      OUT     M7368
2590  LD      X1B35
      AND     M3050
      OUT     M7369
2593  LDI     M7363
      ANI     M7364
      ANI     M7365
      ANI     M7366
      ANI     M7367
      ANI     M7368
      INV
      AND     M7361
      OR      M7362
      ANDPI   M7326
      ANI     M7369
      AND     M7360
      OUT     M7362
2607  LDP     M7362
      MPS
      AND     M7364
      MOVP    K10 D7371
      MRD
      AND     M7365
      MOVP    K11 D7371
      MRD
      LD      M7366
      OR      M7367
      OR      M7363
      ANB
      MOVP    K8 D7371
      MPP
      AND     M7368
      MOVP    K5 D7371
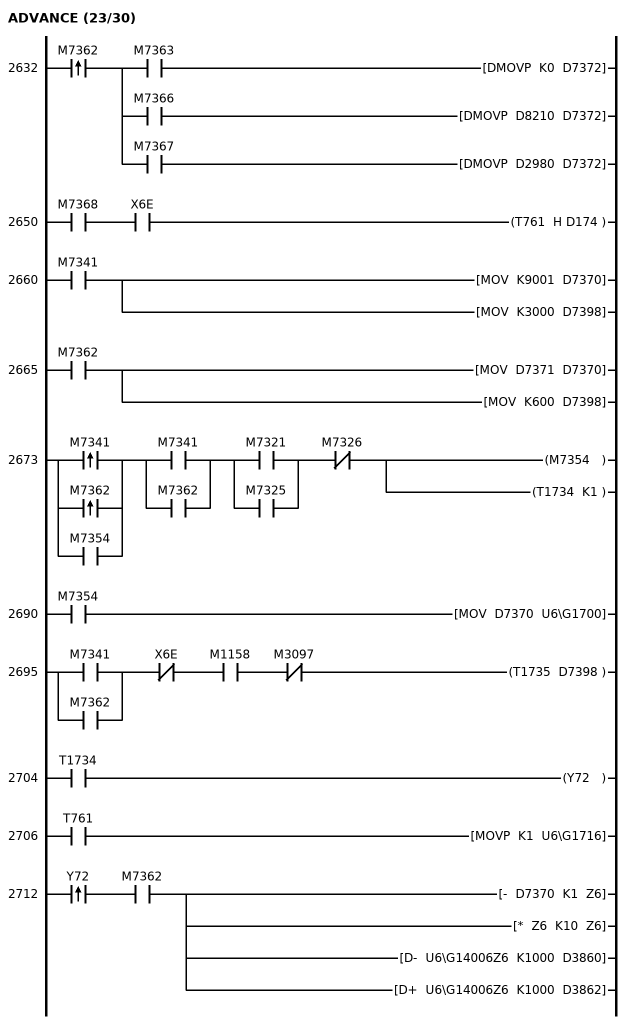
2632  LDP     M7362
      MPS
      AND     M7363
      DMOVP   K0 D7372
      MRD
      AND     M7366
      DMOVP   D8210 D7372
      MPP
      AND     M7367
      DMOVP   D2980 D7372
2650  LD      M7368
      AND     X6E
      OUTH    T761 D174
; 
; 
; 
; 
2660  LD      M7341
      MOV     K9001 D7370
      MOV     K3000 D7398
2665  LD      M7362
      MOV     D7371 D7370
      MOV     K600 D7398
; 
; 
; 
2673  LDP     M7341
      ORP     M7362
      OR      M7354
      LD      M7341
      OR      M7362
      ANB
      LD      M7321
      OR      M7325
      ANB
      ANI     M7326
      OUT     M7354
      OUT     T1734 K1
2690  LD      M7354
      MOV     D7370 U6\G1700
2695  LD      M7341
      OR      M7362
      ANI     X6E
      AND     M1158
      ANI     M3097
      OUT     T1735 D7398
2704  LD      T1734
      OUT     Y72
2706  LD      T761
      MOVP    K1 U6\G1716
2712  LDP     Y72
      AND     M7362
      -       D7370 K1 Z6
      *       Z6 K10 Z6
      D-      U6\G14006Z6 K1000 D3860
      D+      U6\G14006Z6 K1000 D3862
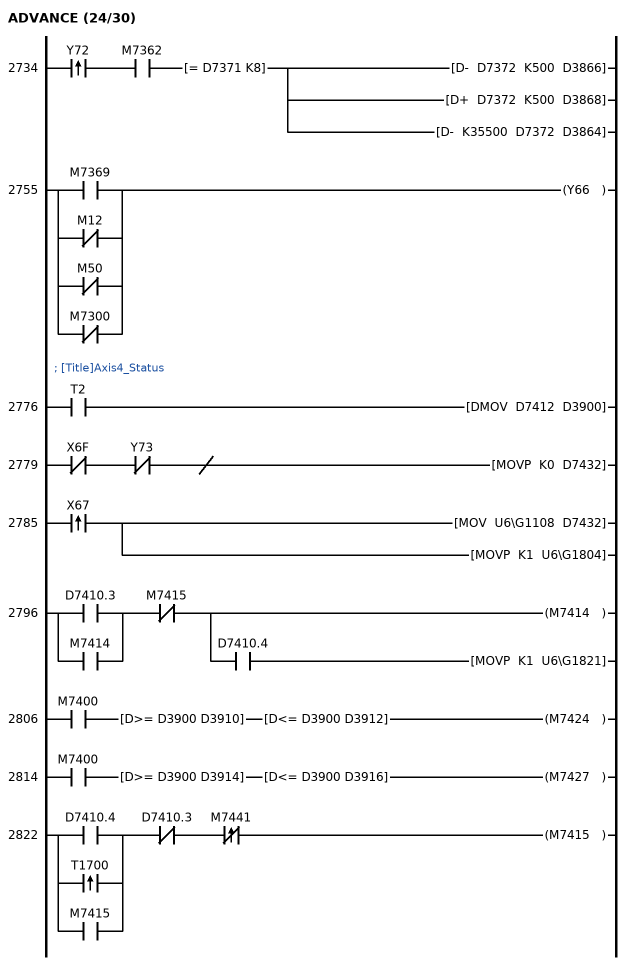
2734  LDP     Y72
      AND     M7362
      AND=    D7371 K8
      D-      D7372 K500 D3866
      D+      D7372 K500 D3868
      D-      K35500 D7372 D3864
; 
; 
; 
2755  LD      M7369
      ORI     M12
      ORI     M50
      ORI     M7300
      OUT     Y66
; 
; 
; [Title]Axis4_Status
; 
; 
2776  LD      T2
      DMOV    D7412 D3900
2779  LDI     X6F
      ANI     Y73
      INV
      MOVP    K0 D7432
2785  LDP     X67
      MOV     U6\G1108 D7432
      MOVP    K1 U6\G1804
2796  LD      D7410.3
      OR      M7414
      ANI     M7415
      OUT     M7414
      AND     D7410.4
      MOVP    K1 U6\G1821
2806  LD      M7400
      ANDD>=  D3900 D3910
      ANDD<=  D3900 D3912
      OUT     M7424
2814  LD      M7400
      ANDD>=  D3900 D3914
      ANDD<=  D3900 D3916
      OUT     M7427
2822  LD      D7410.4
      ORP     T1700
      OR      M7415
      ANI     D7410.3
      ANDPI   M7441
      OUT     M7415
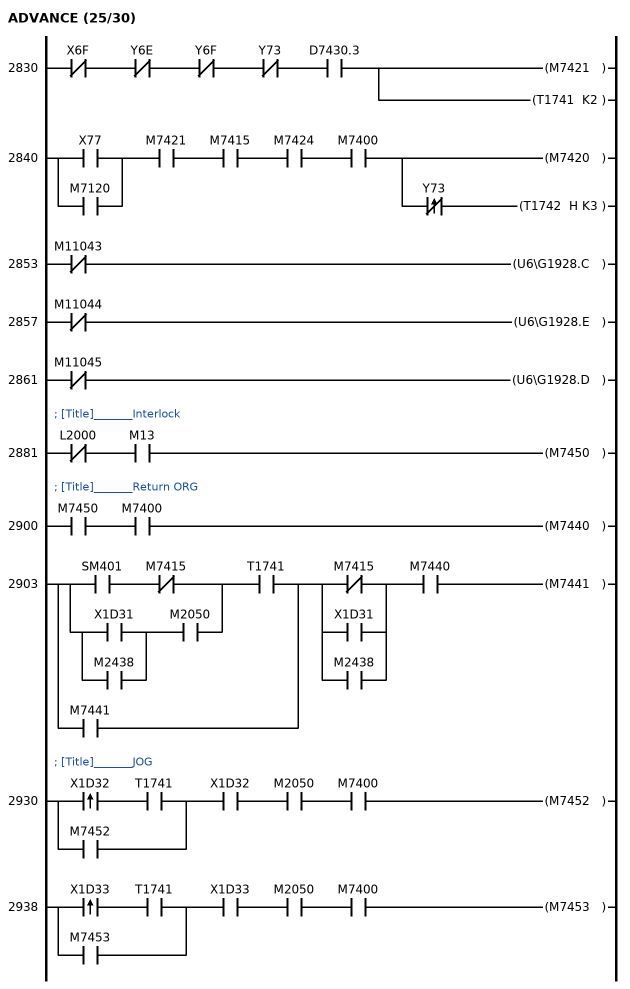
2830  LDI     X6F
      ANI     Y6E
      ANI     Y6F
      ANI     Y73
      AND     D7430.3
      OUT     M7421
      OUT     T1741 K2
2840  LD      X77
      OR      M7120
      AND     M7421
      AND     M7415
      AND     M7424
      AND     M7400
      OUT     M7420
      ANDPI   Y73
      OUTH    T1742 K3
2853  LDI     M11043
      OUT     U6\G1928.C
2857  LDI     M11044
      OUT     U6\G1928.E
2861  LDI     M11045
      OUT     U6\G1928.D
; 
; [Title]_______Interlock
; 
2881  LDI     L2000
      AND     M13
      OUT     M7450
; 
; [Title]_______Return ORG
; 
2900  LD      M7450
      AND     M7400
      OUT     M7440
2903  LD      SM401
      ANI     M7415
      LD      X1D31
      OR      M2438
      AND     M2050
      ORB
      AND     T1741
      OR      M7441
      LDI     M7415
      OR      X1D31
      OR      M2438
      ANB
      AND     M7440
      OUT     M7441
; 
; [Title]_______JOG
; 
2930  LDP     X1D32
      AND     T1741
      OR      M7452
      AND     X1D32
      AND     M2050
      AND     M7400
      OUT     M7452
2938  LDP     X1D33
      AND     T1741
      OR      M7453
      AND     X1D33
      AND     M2050
      AND     M7400
      OUT     M7453
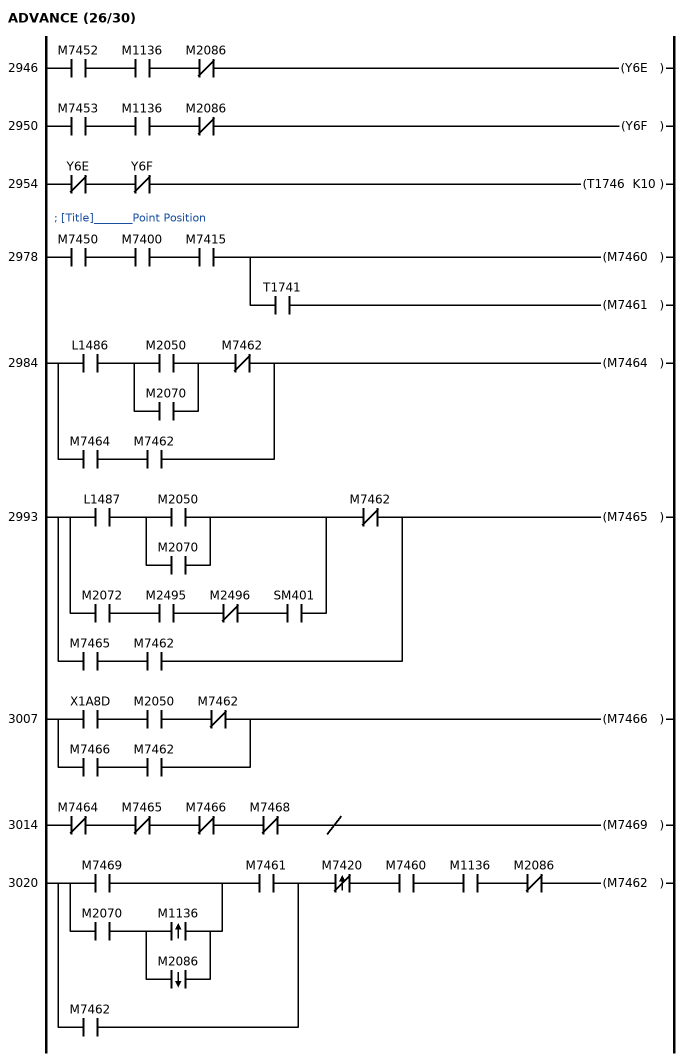
2946  LD      M7452
      AND     M1136
      ANI     M2086
      OUT     Y6E
2950  LD      M7453
      AND     M1136
      ANI     M2086
      OUT     Y6F
2954  LDI     Y6E
      ANI     Y6F
      OUT     T1746 K10
; 
; [Title]_______Point Position
; 
2978  LD      M7450
      AND     M7400
      AND     M7415
      OUT     M7460
      AND     T1741
      OUT     M7461
2984  LD      L1486
      LD      M2050
      OR      M2070
      ANB
      ANI     M7462
      LD      M7464
      AND     M7462
      ORB
      OUT     M7464
2993  LD      L1487
      LD      M2050
      OR      M2070
      ANB
      LD      M2072
      AND     M2495
      ANI     M2496
      AND     SM401
      ORB
      ANI     M7462
      LD      M7465
      AND     M7462
      ORB
      OUT     M7465
3007  LD      X1A8D
      AND     M2050
      ANI     M7462
      LD      M7466
      AND     M7462
      ORB
      OUT     M7466
3014  LDI     M7464
      ANI     M7465
      ANI     M7466
      ANI     M7468
      INV
      OUT     M7469
3020  LD      M7469
      LD      M2070
      LDP     M1136
      ORF     M2086
      ANB
      ORB
      AND     M7461
      OR      M7462
      ANDPI   M7420
      AND     M7460
      AND     M1136
      ANI     M2086
      OUT     M7462
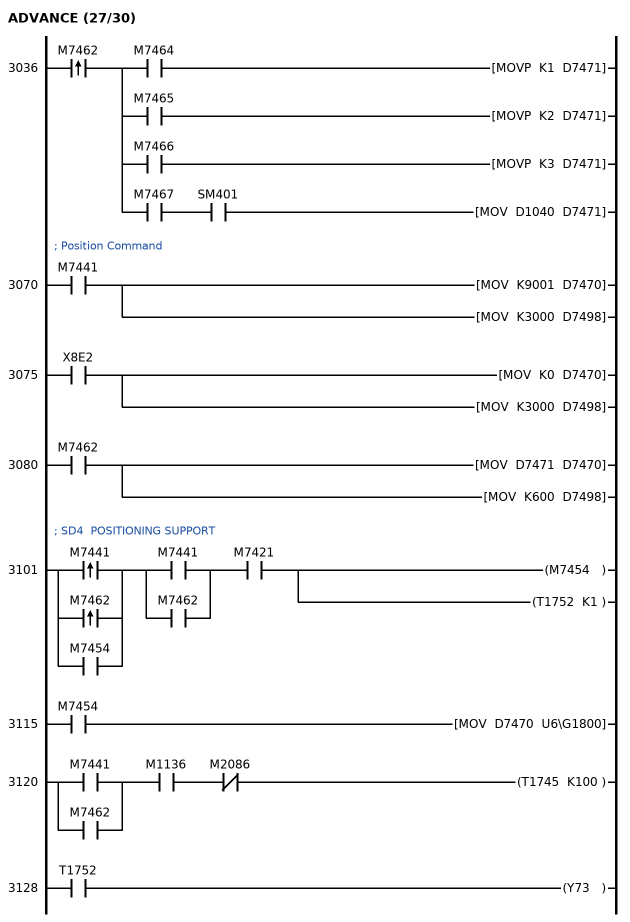
3036  LDP     M7462
      MPS
      AND     M7464
      MOVP    K1 D7471
      MRD
      AND     M7465
      MOVP    K2 D7471
      MRD
      AND     M7466
      MOVP    K3 D7471
      MPP
      AND     M7467
      AND     SM401
      MOV     D1040 D7471
; 
; Position Command
; 
3070  LD      M7441
      MOV     K9001 D7470
      MOV     K3000 D7498
3075  LD      X8E2
      MOV     K0 D7470
      MOV     K3000 D7498
3080  LD      M7462
      MOV     D7471 D7470
      MOV     K600 D7498
; 
; SD4  POSITIONING SUPPORT
; 
3101  LDP     M7441
      ORP     M7462
      OR      M7454
      LD      M7441
      OR      M7462
      ANB
      AND     M7421
      OUT     M7454
      OUT     T1752 K1
3115  LD      M7454
      MOV     D7470 U6\G1800
3120  LD      M7441
      OR      M7462
      AND     M1136
      ANI     M2086
      OUT     T1745 K100
3128  LD      T1752
      OUT     Y73
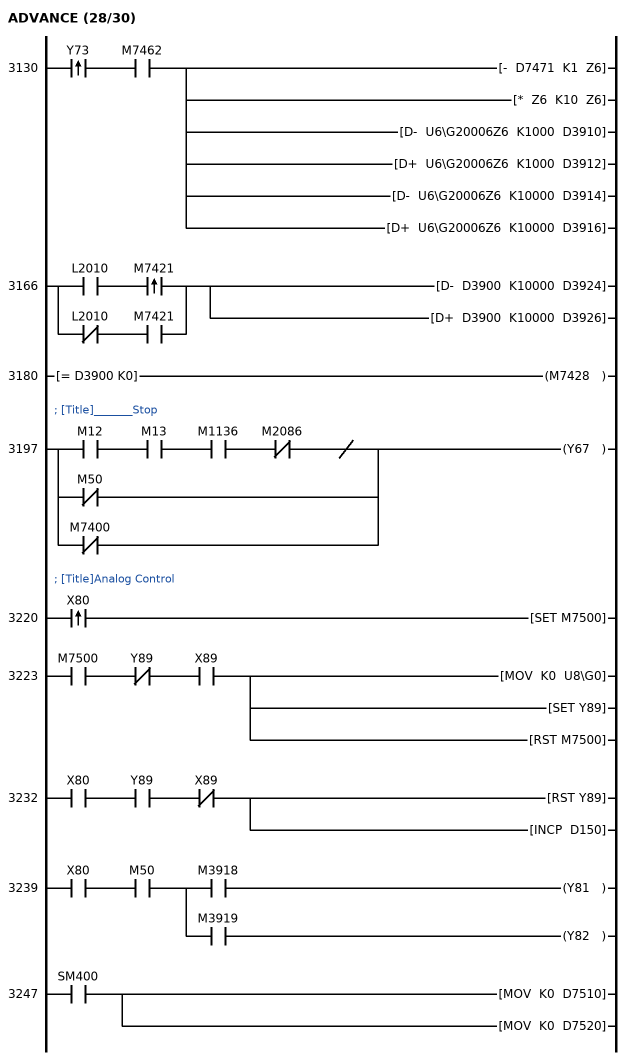
3130  LDP     Y73
      AND     M7462
      -       D7471 K1 Z6
      *       Z6 K10 Z6
      D-      U6\G20006Z6 K1000 D3910
      D+      U6\G20006Z6 K1000 D3912
      D-      U6\G20006Z6 K10000 D3914
      D+      U6\G20006Z6 K10000 D3916
3166  LD      L2010
      ANDP    M7421
      LDI     L2010
      AND     M7421
      ORB
      D-      D3900 K10000 D3924
      D+      D3900 K10000 D3926
3180  LD=     D3900 K0
      OUT     M7428
; 
; [Title]_______Stop
; 
3197  LD      M12
      AND     M13
      AND     M1136
      ANI     M2086
      INV
      ORI     M50
      ORI     M7400
      OUT     Y67
; 
; [Title]Analog Control
; 
3220  LDP     X80
      SET     M7500
3223  LD      M7500
      ANI     Y89
      AND     X89
      MOV     K0 U8\G0
      SET     Y89
      RST     M7500
3232  LD      X80
      AND     Y89
      ANI     X89
      RST     Y89
      INCP    D150
3239  LD      X80
      AND     M50
      MPS
      AND     M3918
      OUT     Y81
      MPP
      AND     M3919
      OUT     Y82
3247  LD      SM400
      MOV     K0 D7510
      MOV     K0 D7520
